Staubli VAL3: vecMax.pgx

public program vecMax(num& x_nInput[], num& x_nResult)
  local num l_nElement
  local num l_nMax
begin

  l_nMax = -999999
  for l_nElement = 0 to size(x_nInput)-1
    l_nMax = max(l_nMax, x_nInput[l_nElement])
  endFor

  x_nResult = l_nMax

end
